// LMC_PacDrive/Application/TemplateFullProgrammingFramework/Visualization/Windows/VIS_Modules
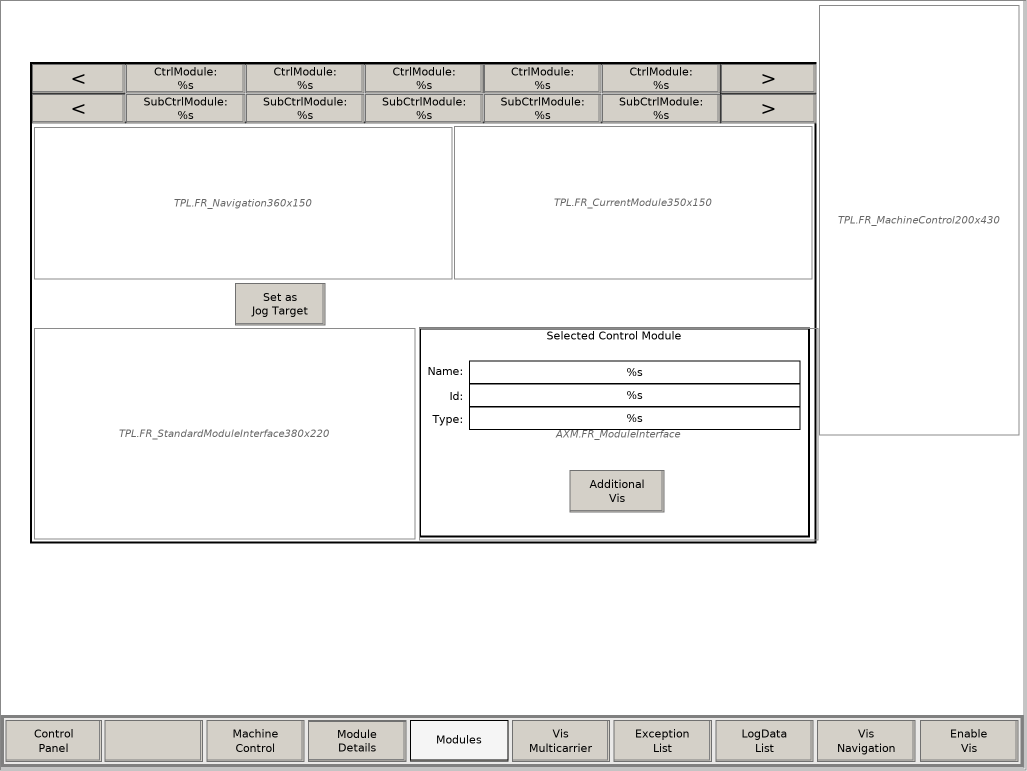
VISUALIZATION VIS_Modules  // 1027x771
    Frame (0,0 1024x768)
        shows TPL.FR_Nav1024x768(i_sTitle := 'Template: Modules')
    Frame (1,715 1024x54)
        shows FR_NavigationButtons()
    Rectangle (30,62 786x481)
    Rectangle (30,63 786x60)
    Button (602,64 118x29), "EQModule: %s", tooltip "%s", text variable: SR_VisControl.vpq_audiIdModuleList[5], colour toggle: SR_VisControl.vpq_axActiveModuleList[5], invisible if: SR_VisControl.vpq_axDisableModuleList[5] OR SR_VisControl.vpq_axIdModuleListValid[5] = FALSE, input disabled if: SR_VisControl.vpq_axDisableModuleList[5]
        p4168582468: SR_VisControl.vpq_asNameModuleList[5]
        toggle SR_VisControl.vpiq_axModuleList[5]
    Button (483,64 118x29), "EQModule: %s", tooltip "%s", text variable: SR_VisControl.vpq_audiIdModuleList[4], colour toggle: SR_VisControl.vpq_axActiveModuleList[4], invisible if: SR_VisControl.vpq_axDisableModuleList[4] OR SR_VisControl.vpq_axIdModuleListValid[4] = FALSE, input disabled if: SR_VisControl.vpq_axDisableModuleList[4]
        p4168582468: SR_VisControl.vpq_asNameModuleList[4]
        toggle SR_VisControl.vpiq_axModuleList[4]
    Button (365,64 118x29), "EQModule: %s", tooltip "%s", text variable: SR_VisControl.vpq_audiIdModuleList[3], colour toggle: SR_VisControl.vpq_axActiveModuleList[3], invisible if: SR_VisControl.vpq_axDisableModuleList[3] OR SR_VisControl.vpq_axIdModuleListValid[3] = FALSE, input disabled if: SR_VisControl.vpq_axDisableModuleList[3]
        p4168582468: SR_VisControl.vpq_asNameModuleList[3]
        toggle SR_VisControl.vpiq_axModuleList[3]
    Button (246,64 118x29), "EQModule: %s", tooltip "%s", text variable: SR_VisControl.vpq_audiIdModuleList[2], colour toggle: SR_VisControl.vpq_axActiveModuleList[2], invisible if: SR_VisControl.vpq_axDisableModuleList[2] OR SR_VisControl.vpq_axIdModuleListValid[2] = FALSE, input disabled if: SR_VisControl.vpq_axDisableModuleList[2]
        p4168582468: SR_VisControl.vpq_asNameModuleList[2]
        toggle SR_VisControl.vpiq_axModuleList[2]
    Button (126,64 119x29), "EQModule: %s", tooltip "%s", text variable: SR_VisControl.vpq_audiIdModuleList[1], colour toggle: SR_VisControl.vpq_axActiveModuleList[1], invisible if: SR_VisControl.vpq_axDisableModuleList[1] OR SR_VisControl.vpq_axIdModuleListValid[1] = FALSE, input disabled if: SR_VisControl.vpq_axDisableModuleList[1]
        p4168582468: SR_VisControl.vpq_asNameModuleList[1]
        toggle SR_VisControl.vpiq_axModuleList[1]
    Button (126,94 119x29), "SubEQModule: %s", tooltip "%s", text variable: SR_VisControl.vpq_audiIdSubModuleList[1], colour toggle: SR_VisControl.vpq_axActiveSubModuleList[1], invisible if: SR_VisControl.vpq_axDisableSubModuleList[1] OR SR_VisControl.vpq_axIdSubModuleListValid[1] = FALSE, input disabled if: SR_VisControl.vpq_axDisableSubModuleList[1]
        p4168582468: SR_VisControl.vpq_asNameSubModuleList[1]
        toggle SR_VisControl.vpiq_axSubModuleList[1]
    Button (246,94 118x29), "SubEQModule: %s", tooltip "%s", text variable: SR_VisControl.vpq_audiIdSubModuleList[2], colour toggle: SR_VisControl.vpq_axActiveSubModuleList[2], invisible if: SR_VisControl.vpq_axDisableSubModuleList[2] OR SR_VisControl.vpq_axIdSubModuleListValid[2] = FALSE, input disabled if: SR_VisControl.vpq_axDisableSubModuleList[2]
        p4168582468: SR_VisControl.vpq_asNameSubModuleList[2]
        toggle SR_VisControl.vpiq_axSubModuleList[2]
    Button (365,94 118x29), "SubEQModule: %s", tooltip "%s", text variable: SR_VisControl.vpq_audiIdSubModuleList[3], colour toggle: SR_VisControl.vpq_axActiveSubModuleList[3], invisible if: SR_VisControl.vpq_axDisableSubModuleList[3] OR SR_VisControl.vpq_axIdSubModuleListValid[3] = FALSE, input disabled if: SR_VisControl.vpq_axDisableSubModuleList[3]
        p4168582468: SR_VisControl.vpq_asNameSubModuleList[3]
        toggle SR_VisControl.vpiq_axSubModuleList[3]
    Button (484,94 117x29), "SubEQModule: %s", tooltip "%s", text variable: SR_VisControl.vpq_audiIdSubModuleList[4], colour toggle: SR_VisControl.vpq_axActiveSubModuleList[4], invisible if: SR_VisControl.vpq_axDisableSubModuleList[4] OR SR_VisControl.vpq_axIdSubModuleListValid[4] = FALSE, input disabled if: SR_VisControl.vpq_axDisableSubModuleList[4]
        p4168582468: SR_VisControl.vpq_asNameSubModuleList[4]
        toggle SR_VisControl.vpiq_axSubModuleList[4]
    Button (602,94 118x29), "SubEQModule: %s", tooltip "%s", text variable: SR_VisControl.vpq_audiIdSubModuleList[5], colour toggle: SR_VisControl.vpq_axActiveSubModuleList[5], invisible if: SR_VisControl.vpq_axDisableSubModuleList[5] OR SR_VisControl.vpq_axIdSubModuleListValid[5] = FALSE, input disabled if: SR_VisControl.vpq_axDisableSubModuleList[5]
        p4168582468: SR_VisControl.vpq_asNameSubModuleList[5]
        toggle SR_VisControl.vpiq_axSubModuleList[5]
    Rectangle (720,93 95x29), ">"
    Rectangle (720,63 95x30), ">"
    Button (721,64 95x29), ">", invisible if: SR_VisControl.vpq_xDisableModuleListUp, input disabled if: SR_VisControl.vpq_xDisableModuleListUp
        toggle SR_VisControl.vpiq_xModuleListUp
    Button (721,94 95x29), ">", invisible if: SR_VisControl.vpq_xDisableSubModuleListUp, input disabled if: SR_VisControl.vpq_xDisableSubModuleListUp
        toggle SR_VisControl.vpiq_xSubModuleListUp
    Rectangle (31,93 94x29), "<"
    Rectangle (31,64 94x30), "<"
    Button (32,64 93x29), "<", invisible if: SR_VisControl.vpq_xDisableModuleListDown, input disabled if: SR_VisControl.vpq_xDisableModuleListDown
        toggle SR_VisControl.vpiq_xModuleListDown
    Button (32,94 93x29), "<", invisible if: SR_VisControl.vpq_xDisableSubModuleListDown, input disabled if: SR_VisControl.vpq_xDisableSubModuleListDown
        toggle SR_VisControl.vpiq_xSubModuleListDown
    Button (235,283 90x42), "Set as Jog Target", colour toggle: SR_VisControl.vpq_xCurrentIsJogTarget, invisible if: SR_VisControl.vpq_xButtonSetJogTargetInvisible
        tap SR_VisControl.vpiq_xButtonSetCurrentAsJogTarget
    Frame (34,127 418x152)
        shows TPL.FR_Navigation360x150(i_sNameNavRight := SR_VisControl.vpq_sNameNavRight, i_sNameNavUp := SR_VisControl.vpq_sNameNavUp, i_sNameNavLeft := SR_VisControl.vpq_sNameNavLeft, i_sNameNavDown := SR_VisControl.vpq_sNameNavDown, i_xEnableNavUp := SR_VisControl.vpq_xEnableNavUp, i_xEnableNavLeft := SR_VisControl.vpq_xEnableNavLeft, i_xEnableNavRight := SR_VisControl.vpq_xEnableNavRight, i_xEnableNavDown := SR_VisControl.vpq_xEnableNavDown, iq_xNavUp := SR_VisControl.vpiq_xNavUp, iq_xNavLeft := SR_VisControl.vpiq_xNavLeft, iq_xNavRight := SR_VisControl.vpiq_xNavRight, iq_xNavDown := SR_VisControl.vpiq_xNavDown)
    Frame (454,126 358x153)
        shows TPL.FR_CurrentModule350x150(i_stCurrentModuleStandardItf := SR_VisControl.vpq_stCurrentModuleStandardInterface)
        p2332068554: SR_VisControl.stCurrentModuleStandardInterface
        p427866952: SR_VisControl.stCurrentModuleStandardInterface
        p2190627833: SR_VisControl.vpq_stCurrentModuleStandardInterface
    Button (126,64 119x29), "CtrlModule: %s", tooltip "%s", text variable: SR_VisControl.vpq_asControlModuleButtonName[1], colour toggle: SR_VisControl.vpq_axControlModuleActive[1], invisible if: SR_VisControl.vpq_axControlModuleValid[1]=FALSE
        p4168582468: SR_VisControl.vpq_asToolTipControlModuleList[1]
        toggle SR_VisControl.vpiq_axControlModuleList[1]
    Button (246,64 118x29), "CtrlModule: %s", tooltip "%s", text variable: SR_VisControl.vpq_asControlModuleButtonName[2], colour toggle: SR_VisControl.vpq_axControlModuleActive[2], invisible if: SR_VisControl.vpq_axControlModuleValid[2]=FALSE
        p4168582468: SR_VisControl.vpq_asToolTipControlModuleList[2]
        toggle SR_VisControl.vpiq_axControlModuleList[2]
    Button (365,64 118x29), "CtrlModule: %s", tooltip "%s", text variable: SR_VisControl.vpq_asControlModuleButtonName[3], colour toggle: SR_VisControl.vpq_axControlModuleActive[3], invisible if: SR_VisControl.vpq_axControlModuleValid[3]=FALSE
        p4168582468: SR_VisControl.vpq_asToolTipControlModuleList[3]
        toggle SR_VisControl.vpiq_axControlModuleList[3]
    Button (484,64 117x29), "CtrlModule: %s", tooltip "%s", text variable: SR_VisControl.vpq_asControlModuleButtonName[4], colour toggle: SR_VisControl.vpq_axControlModuleActive[4], invisible if: SR_VisControl.vpq_axControlModuleValid[4]=FALSE
        p4168582468: SR_VisControl.vpq_asToolTipControlModuleList[4]
        toggle SR_VisControl.vpiq_axControlModuleList[4]
    Button (602,64 118x29), "CtrlModule: %s", tooltip "%s", text variable: SR_VisControl.vpq_asControlModuleButtonName[5], colour toggle: SR_VisControl.vpq_axControlModuleActive[5], invisible if: SR_VisControl.vpq_axControlModuleValid[5]=FALSE
        p4168582468: SR_VisControl.vpq_asToolTipControlModuleList[5]
        toggle SR_VisControl.vpiq_axControlModuleList[5]
    Button (126,94 119x29), "SubCtrlModule: %s", tooltip "%s", text variable: SR_VisControl.vpq_asSubControlModuleButtonName[1], colour toggle: SR_VisControl.vpq_axSubControlModuleActive[1], invisible if: SR_VisControl.vpq_axSubControlModuleValid[1]=FALSE
        p4168582468: SR_VisControl.vpq_asToolTipSubControlModuleList[1]
        toggle SR_VisControl.vpiq_axSubControlModuleList[1]
    Button (246,94 118x29), "SubCtrlModule: %s", tooltip "%s", text variable: SR_VisControl.vpq_asSubControlModuleButtonName[2], colour toggle: SR_VisControl.vpq_axSubControlModuleActive[2], invisible if: SR_VisControl.vpq_axSubControlModuleValid[2]=FALSE
        p4168582468: SR_VisControl.vpq_asToolTipSubControlModuleList[2]
        toggle SR_VisControl.vpiq_axSubControlModuleList[2]
    Button (365,94 118x29), "SubCtrlModule: %s", tooltip "%s", text variable: SR_VisControl.vpq_asSubControlModuleButtonName[3], colour toggle: SR_VisControl.vpq_axSubControlModuleActive[3], invisible if: SR_VisControl.vpq_axSubControlModuleValid[3]=FALSE
        p4168582468: SR_VisControl.vpq_asToolTipSubControlModuleList[3]
        toggle SR_VisControl.vpiq_axSubControlModuleList[3]
    Button (484,94 117x29), "SubCtrlModule: %s", tooltip "%s", text variable: SR_VisControl.vpq_asSubControlModuleButtonName[4], colour toggle: SR_VisControl.vpq_axSubControlModuleActive[4], invisible if: SR_VisControl.vpq_axSubControlModuleValid[4]=FALSE
        p4168582468: SR_VisControl.vpq_asToolTipSubControlModuleList[4]
        toggle SR_VisControl.vpiq_axSubControlModuleList[4]
    Button (602,94 118x29), "SubCtrlModule: %s", tooltip "%s", text variable: SR_VisControl.vpq_asSubControlModuleButtonName[5], colour toggle: SR_VisControl.vpq_axSubControlModuleActive[5], invisible if: SR_VisControl.vpq_axSubControlModuleValid[5]=FALSE
        p4168582468: SR_VisControl.vpq_asToolTipSubControlModuleList[5]
        toggle SR_VisControl.vpiq_axSubControlModuleList[5]
    Frame (418,327 394x212), invisible if: SR_VisControl.vpq_udiActiveControlModuleNumber <> 0
        shows FR_OtherModuleTypes()
    Frame (418,327 394x212), invisible if: SR_VisControl.vpq_udiActiveControlModuleNumber = 0
        shows FR_ControlModuleTypes(i_sControlModuleName := SR_VisControl.stCurrentControlModuleStandardInterface.sControlModuleName, i_diControlModuleNumber := TO_DINT(SR_VisControl.stCurrentControlModuleStandardInterface.udiControlModuleNumber), i_diControlModuleType := TO_DINT(SR_VisControl.stCurrentControlModuleStandardInterface.udiControlModuleType))
        p159172089: SR_VisControl.IFB_AxisModuleVisController
        p2210332906: SR_VisControl.IFB_AxisModuleVisController.iPaneSelect
    Frame (34,328 381x211)
        shows TPL.FR_StandardModuleInterface380x220(i_stCurrentModuleStandardItf := SR_VisControl.vpq_stCurrentModuleStandardInterface, i_sCurrentModuleReaction := SR_VisControl.vpq_sCurrentModuleReaction, i_udiModuleReactionIndexMin := SR_VisControl.vpq_udiModuleReactionIndexMin, i_axModuleReaction := SR_VisControl.vpq_axModuleReaction, i_udiNumberOfReactions := TPL.Gc_udiMaxNumberOfReactions, iq_xModuleReactionDown := SR_VisControl.vpiq_xModuleReactionDown, iq_xModuleReactionUp := SR_VisControl.vpiq_xModuleReactionUp, iq_diStartStepToSet := SR_VisControl.vpiq_diStartStepToSet, iq_diCmdToSet := SR_VisControl.vpiq_diCmdToSet, iq_xEnableModuleClicked := SR_VisControl.vpiq_xEnableModuleClicked, iq_xSetCmdClicked := SR_VisControl.vpiq_xSetCmdClicked, iq_fbVisContExHandling := SR_VisControl.vpiq_fbVisContExHandling)
        p1094400588: SR_VisControl.IFB_AxisModuleVisController.xCurrentIsOfMyType
        p3339340907: 'Vis_ModuleError'
        p1029787830: SR_VisControl.vpiq_fbVisContExHandling
        p2258115317: SR_VisControl.iModuleErrorReactionIndexMin
        p2777435286: SR_VisControl.axModuleErrorReaction
        p214250784: TPC_Gc_diMaxNumberOfErrorReactions
        p311732222: SR_VisControl.stCurrentModuleStandardInterface
        p640132070: SR_VisControl.xModuleErrorReactionDown
        p4234372197: SR_VisControl.xModuleErrorReactionUp
        p2938682392: SR_VisControl.xEnableModule_Clicked
        p3592490199: SR_VisControl.xSetCmd_Clicked
        p2560461379: SR_VisControl.diStartStepToSet
        p2307280719: SR_VisControl.stCurrentModuleStandardInterface
        p2190627833: SR_VisControl.vpq_stCurrentModuleStandardInterface
    Frame (419,328 399x212), invisible if: SR_VisControl.vpq_stCurrentModuleStandardInterface.q_dwModuleType <> 3
        shows AXM.FR_ModuleInterface(iq_fbAxisModuleVisController := SR_VisControl.vpiq_fbAxisModuleVisController)
        p159172089: SR_VisControl.IFB_AxisModuleVisController
        p2210332906: SR_VisControl.IFB_AxisModuleVisController.iPaneSelect
        p856915466: SR_VisControl.stCurrentControlModuleStandardInterface.udiControlModuleNumber
        p2344652976: SR_VisControl.stCurrentControlModuleStandardInterface.udiControlModuleType
        p467735965: SR_VisControl.stCurrentControlModuleStandardInterface.sControlModuleName
    Button (308,721 98x40), "Module Details"
        OnMouseClick:  Assign=VIS_ModuleDetails, Type=Assignment
    Rectangle (410,720 98x40), "Modules"
    Frame (819,5 200x430), invisible if: NOT SR_VisControl.vpiq_xShowControlFrame
        shows TPL.FR_MachineControl200x430(i_stMachineItf := SR_VisControl.vpq_stMachineInterface, i_xPrepareActive := G_xPrepareActive, i_xAutoActive := G_xAutoActive, i_xBrakeReleaseActive := G_xBrakeReleaseActive, i_xJogMachineActive := G_xJogMachineActive, i_xManualActive := G_xManualActive, i_xException := SR_VisControl.vpq_xMachineInException, i_dwDiagQuitColor := SR_VisControl.vpq_dwDiagQuitColor, iq_iPositionX := SR_VisControl.vpiq_iPositionX, iq_iPositionY := SR_VisControl.vpiq_iPositionY, iq_xEmergencyEpas := G_xEmergencyEpas, iq_xStartEpas := G_xStartEpas, iq_xStopEpas := G_xStopEpas, iq_xJogForwEpas := G_xJogForwEpas, iq_xJogBackEpas := G_xJogBackEpas, iq_xDoPrepare := G_xDoPrepare, iq_xDoAuto := G_xDoAuto, iq_xDoBrakeRelease := G_xDoBrakeRelease, iq_xDoJogMachine := G_xDoJogMachine, iq_xDoManual := G_xDoManual, iq_xDiagQuitEpas := G_xDiagQuitEpas)
        p1457045297: SR_VisControl.stMachineInterface.stQ.xError
        p1941967854: g_I_xEmergency_Epas
        p2531571229: g_I_xStart_Epas
        p1511842254: g_I_xStop_Epas
        p745511063: g_I_xJogForw_Epas
        p3518271027: g_I_xJogBack_Epas
        p1982879521: g_I_xErrorQuit_Epas
        p3866886353: SR_VisControl.dwErrorQuitColor
        p1761348311: SR_VisControl.vpq_stMachineInterface
        p3560616238: SR_VisControl.vpiq_iPositionX
        p2738717112: SR_VisControl.vpiq_iPositionY
END_VISUALIZATION

// LMC_PacDrive/Application/TemplateFullProgrammingFramework/Visualization/Windows/VIS_VisNavigation
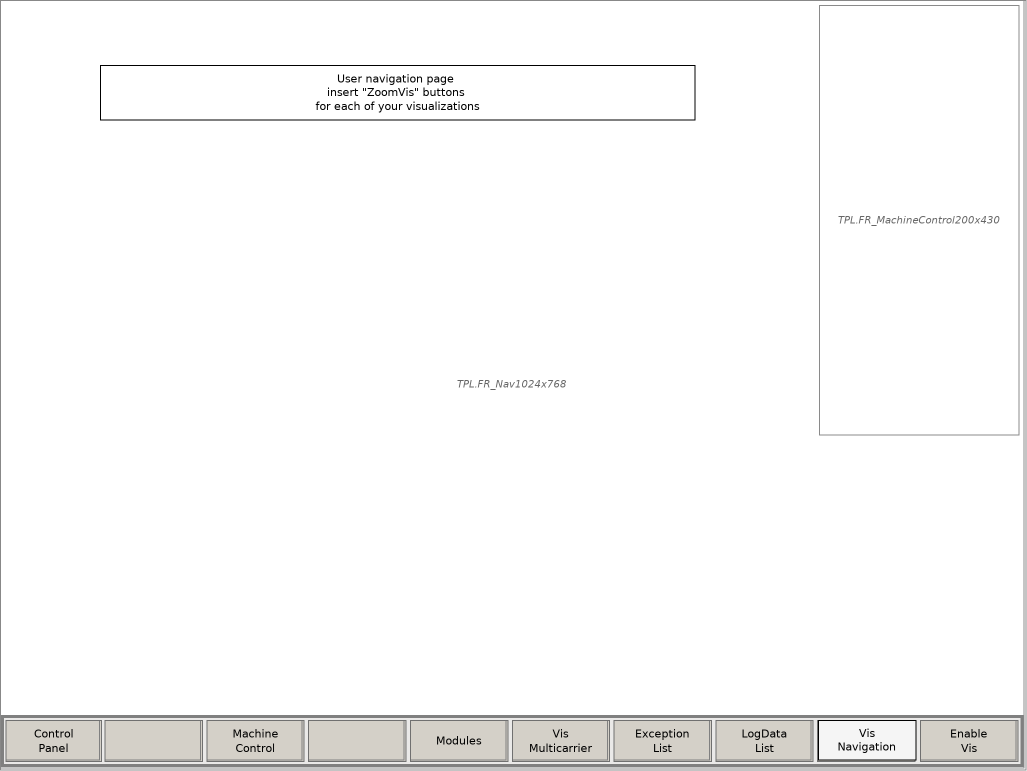
VISUALIZATION VIS_VisNavigation  // 1027x771
    Frame (0,0 1024x768)
        shows TPL.FR_Nav1024x768(i_sTitle := 'Template: Navigation')
    Rectangle (100,65 595x55), "User navigation page insert "ZoomVis" buttons for each of your visualizations"
    Frame (1,715 1024x54)
        shows FR_NavigationButtons()
    Rectangle (818,720 98x40), "Vis Navigation"
    Frame (819,5 200x430), invisible if: NOT SR_VisControl.vpiq_xShowControlFrame
        shows TPL.FR_MachineControl200x430(i_stMachineItf := SR_VisControl.vpq_stMachineInterface, i_xPrepareActive := G_xPrepareActive, i_xAutoActive := G_xAutoActive, i_xBrakeReleaseActive := G_xBrakeReleaseActive, i_xJogMachineActive := G_xJogMachineActive, i_xManualActive := G_xManualActive, i_xException := SR_VisControl.vpq_xMachineInException, i_dwDiagQuitColor := SR_VisControl.vpq_dwDiagQuitColor, iq_iPositionX := SR_VisControl.vpiq_iPositionX, iq_iPositionY := SR_VisControl.vpiq_iPositionY, iq_xEmergencyEpas := G_xEmergencyEpas, iq_xStartEpas := G_xStartEpas, iq_xStopEpas := G_xStopEpas, iq_xJogForwEpas := G_xJogForwEpas, iq_xJogBackEpas := G_xJogBackEpas, iq_xDoPrepare := G_xDoPrepare, iq_xDoAuto := G_xDoAuto, iq_xDoBrakeRelease := G_xDoBrakeRelease, iq_xDoJogMachine := G_xDoJogMachine, iq_xDoManual := G_xDoManual, iq_xDiagQuitEpas := G_xDiagQuitEpas)
        p1457045297: SR_VisControl.stMachineInterface.stQ.xError
        p1941967854: g_I_xEmergency_Epas
        p2531571229: g_I_xStart_Epas
        p1511842254: g_I_xStop_Epas
        p745511063: g_I_xJogForw_Epas
        p3518271027: g_I_xJogBack_Epas
        p1982879521: g_I_xErrorQuit_Epas
        p3866886353: SR_VisControl.dwErrorQuitColor
        p1761348311: SR_VisControl.vpq_stMachineInterface
        p3560616238: SR_VisControl.vpiq_iPositionX
        p2738717112: SR_VisControl.vpiq_iPositionY
END_VISUALIZATION

// LMC_PacDrive/Application/TemplateFullProgrammingFramework/EquipmentModules/MulticarrierModule/Multicarrier Stations/AutomaticMode/Vis_Auto
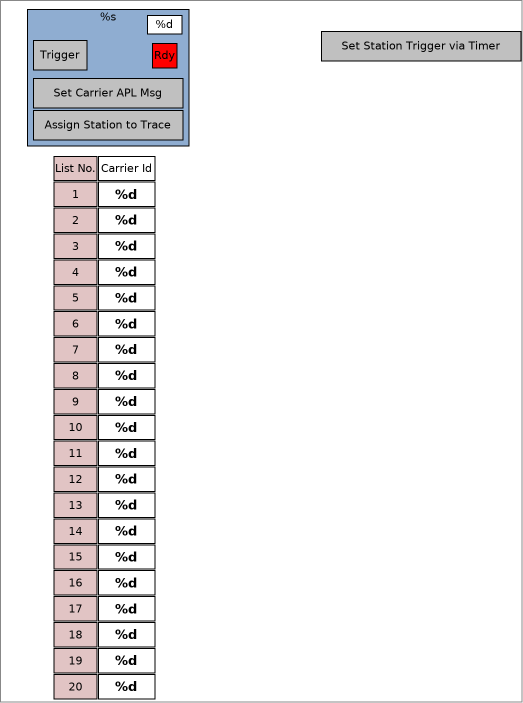
VISUALIZATION Vis_Auto  // 523x703
    Rectangle (27,9 162x137), "%s", text variable: SR_MultiCarrierModule.fbStation1.sName, input disabled if: NOT SR_MainMachine.xActAuto
    Rectangle (33,40 54x30), "Trigger", input disabled if: NOT SR_MainMachine.xActAuto
        tap SR_MulticarrierModule.stStation1.xTrigger
    Rectangle (147,15 35x19), "%d", tooltip "Total number of Carriers in Station", text variable: SR_MulticarrierModule.fbStation1.udiNumberOfCarriersInStationTotal, input disabled if: NOT SR_MainMachine.xActAuto
    Frame (53,156 104x545), input disabled if: NOT SR_MainMachine.xActAuto
        shows FR_List(iq_uiCarrierIndex := SR_MulticarrierModule.fbStation1.raudiCarrierIndexArray)
    Rectangle (33,110 150x30), "Assign Station to Trace", colour toggle: SR_MultiCarrierModule.etTraceSource = ET_TraceSource.Station1, input disabled if: NOT SR_MainMachine.xActAuto
        OnMouseClick: execute { SR_MultiCarrierModule.etTraceSource := ET_TraceSource.Station1; }
    Rectangle (33,78 150x30), "Set Carrier APL Msg", colour toggle: SR_MulticarrierModule.stStation1.xApplicationLoggerEntriesActive, input disabled if: NOT SR_MainMachine.xActAuto
        toggle SR_MulticarrierModule.stStation1.xApplicationLoggerEntriesActive
    RoundedRectangle (152,43 25x25), "Rdy", colour toggle: SR_MulticarrierModule.fbStation1.xStationReadyForJob, input disabled if: NOT SR_MainMachine.xActAuto
    Rectangle (321,31 200x30), "Set Station Trigger via Timer", input disabled if: NOT SR_MainMachine.xActAuto
        toggle SR_MultiCarrierModule.xSetStationTriggerViaTimer
END_VISUALIZATION

// LMC_PacDrive/Application/TemplateFullProgrammingFramework/EquipmentModules/MulticarrierModule/Multicarrier Stations/AutomaticMode/Vis_StationCopyMaster
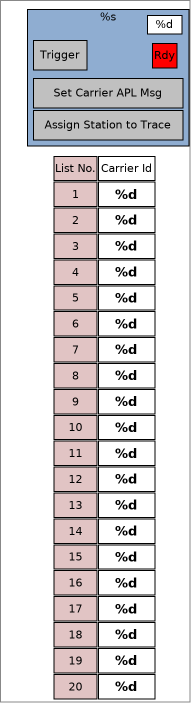
VISUALIZATION Vis_StationCopyMaster  // 191x703
    Rectangle (27,9 162x137), "%s", text variable: SR_MultiCarrierModule.fbStation1.sName, input disabled if: NOT SR_MainMachine.xActAuto
    Rectangle (33,40 54x30), "Trigger", input disabled if: NOT SR_MainMachine.xActAuto
        tap SR_MulticarrierModule.stStation1.xTrigger
    Rectangle (147,15 35x19), "%d", tooltip "Total number of Carriers in Station", text variable: SR_MulticarrierModule.fbStation1.udiNumberOfCarriersInStationTotal, input disabled if: NOT SR_MainMachine.xActAuto
    Frame (53,156 104x545), input disabled if: NOT SR_MainMachine.xActAuto
        shows FR_List(iq_uiCarrierIndex := SR_MultiCarriermodule.fbStation1.raudiCarrierIndexArray)
    Rectangle (33,110 150x30), "Assign Station to Trace", colour toggle: SR_MultiCarrierModule.etTraceSource = ET_TraceSource.Station1, input disabled if: NOT SR_MainMachine.xActAuto
        OnMouseClick: execute { SR_MultiCarrierModule.etTraceSource := ET_TraceSource.Station1; }
    Rectangle (33,78 150x30), "Set Carrier APL Msg", colour toggle: SR_MulticarrierModule.stStation1.xApplicationLoggerEntriesActive, input disabled if: NOT SR_MainMachine.xActAuto
        toggle SR_MulticarrierModule.stStation1.xApplicationLoggerEntriesActive
    RoundedRectangle (152,43 25x25), "Rdy", colour toggle: SR_MulticarrierModule.fbStation1.xStationReadyForJob, input disabled if: NOT SR_MainMachine.xActAuto
END_VISUALIZATION

// LMC_PacDrive/Application/TemplateFullProgrammingFramework/EquipmentModules/MulticarrierModule/Multicarrier Stations/Test Multicarrier/Vis_TestMulticarrier
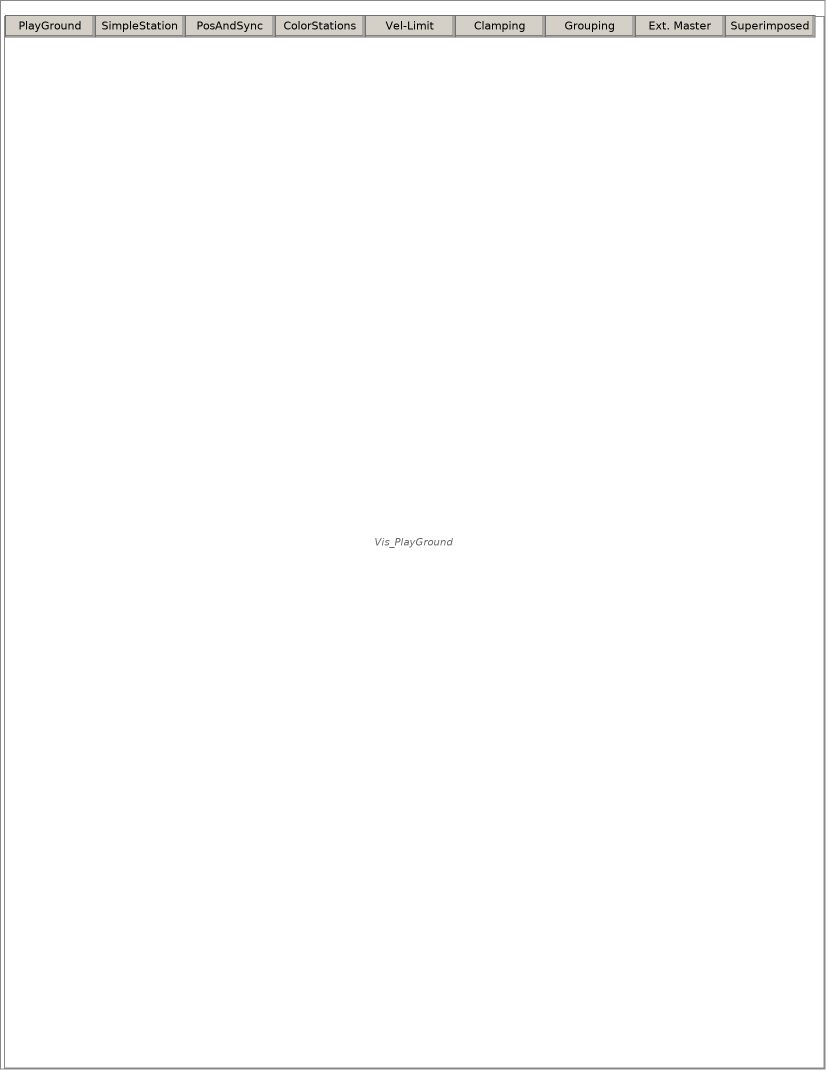
VISUALIZATION Vis_TestMulticarrier  // 826x1070
    TabControl (4,16 820x1052), frame switch variable: SR_CallTestStations.uiSetOpModeTestVis
        shows Vis_PlayGround()
        shows Vis_SimpleStations()
        shows Vis_PosAndSync()
        shows Vis_ColorStations()
        shows Vis_VelLimit()
        shows Vis_ClampingDeclampingStations()
        shows Vis_Grouping()
        shows Vis_ExternalMaster()
        shows Vis_Superimposed()
        [0]: TabTitle=PlayGround
        [1]: TabTitle=SimpleStation
        [2]: TabTitle=PosAndSync
        [3]: TabTitle=ColorStations
        [4]: TabTitle=VelLimit
        [5]: TabTitle=Clamping
        [6]: TabTitle=Grouping
        [7]: TabTitle=Ext. Master
    Button (5,15 90x22), "PlayGround", colour toggle: SR_CallTestStations.uiSetOpModeTestVis = 0
        OnMouseClick: execute { SR_CallTestStations.uiSetOpModeTestVis := 0; }
    Button (95,15 90x22), "SimpleStation", colour toggle: SR_CallTestStations.uiSetOpModeTestVis = 1
        OnMouseClick: execute { SR_CallTestStations.uiSetOpModeTestVis := 1; }
    Button (185,15 90x22), "PosAndSync", colour toggle: SR_CallTestStations.uiSetOpModeTestVis = 2
        OnMouseClick: execute { SR_CallTestStations.uiSetOpModeTestVis := 2; }
    Button (275,15 90x22), "ColorStations", colour toggle: SR_CallTestStations.uiSetOpModeTestVis = 3
        OnMouseClick: execute { SR_CallTestStations.uiSetOpModeTestVis := 3; }
    Button (365,15 90x22), "Vel-Limit", colour toggle: SR_CallTestStations.uiSetOpModeTestVis = 4
        OnMouseClick: execute { SR_CallTestStations.uiSetOpModeTestVis := 4; }
    Button (455,15 90x22), "Clamping", colour toggle: SR_CallTestStations.uiSetOpModeTestVis = 5
        OnMouseClick: execute { SR_CallTestStations.uiSetOpModeTestVis := 5; }
    Button (545,15 90x22), "Grouping", colour toggle: SR_CallTestStations.uiSetOpModeTestVis = 6
        OnMouseClick: execute { SR_CallTestStations.uiSetOpModeTestVis := 6; }
    Button (635,15 90x22), "Ext. Master", colour toggle: SR_CallTestStations.uiSetOpModeTestVis = 7
        OnMouseClick: execute { SR_CallTestStations.uiSetOpModeTestVis := 7; }
    Button (725,15 90x22), "Superimposed", colour toggle: SR_CallTestStations.uiSetOpModeTestVis = 8
        OnMouseClick: execute { SR_CallTestStations.uiSetOpModeTestVis := 8; }
END_VISUALIZATION

(* text list TextList_VisPositions (id | default)
  0 | RefTrackPos
  1 | RefPosition
  2 | Gap in Front
  3 | Dist in Front
  4 | Gap Behind
  5 | Dist Behind
   |  *)
